DATA_BLOCK "S1.CABINET097.ALARM2"   // DB2589
// stored: AutoNumber true, DBAccessibleFromOPCUA true, DBAccessibleFromWebserver true, InstanceOfName BoolToUDInt_Inverted_Filtered, InstanceOfType FB
"BoolToUDInt_Inverted_Filtered "
BEGIN
END_DATA_BLOCK

DATA_BLOCK "S1.CABINET097.WARNING1"   // DB2590
// stored: AutoNumber true, DBAccessibleFromOPCUA true, DBAccessibleFromWebserver true, InstanceOfName BoolToUDInt_Inverted_Filtered, InstanceOfType FB
"BoolToUDInt_Inverted_Filtered "
BEGIN
END_DATA_BLOCK

DATA_BLOCK "S1.CABINET097.WARNING2"   // DB2591
// stored: AutoNumber true, DBAccessibleFromOPCUA true, DBAccessibleFromWebserver true, InstanceOfName BoolToUDInt_Inverted_Filtered, InstanceOfType FB
"BoolToUDInt_Inverted_Filtered "
BEGIN
END_DATA_BLOCK

DATA_BLOCK "S1.CABINET098.ALARM1"   // DB2592
// stored: AutoNumber true, DBAccessibleFromOPCUA true, DBAccessibleFromWebserver true, InstanceOfName BoolToUDInt_Inverted_Filtered, InstanceOfType FB
"BoolToUDInt_Inverted_Filtered "
BEGIN
END_DATA_BLOCK

DATA_BLOCK "S1.CABINET098.ALARM2"   // DB2593
// stored: AutoNumber true, DBAccessibleFromOPCUA true, DBAccessibleFromWebserver true, InstanceOfName BoolToUDInt_Inverted_Filtered, InstanceOfType FB
"BoolToUDInt_Inverted_Filtered "
BEGIN
END_DATA_BLOCK

DATA_BLOCK "S1.CABINET098.WARNING1"   // DB2594
// stored: AutoNumber true, DBAccessibleFromOPCUA true, DBAccessibleFromWebserver true, InstanceOfName BoolToUDInt_Inverted_Filtered, InstanceOfType FB
"BoolToUDInt_Inverted_Filtered "
BEGIN
END_DATA_BLOCK

DATA_BLOCK "S1.CABINET098.WARNING2"   // DB2595
// stored: AutoNumber true, DBAccessibleFromOPCUA true, DBAccessibleFromWebserver true, InstanceOfName BoolToUDInt_Inverted_Filtered, InstanceOfType FB
"BoolToUDInt_Inverted_Filtered "
BEGIN
END_DATA_BLOCK

DATA_BLOCK "S1.CABINET099.ALARM1"   // DB2596
// stored: AutoNumber true, DBAccessibleFromOPCUA true, DBAccessibleFromWebserver true, InstanceOfName BoolToUDInt_Inverted_Filtered, InstanceOfType FB
"BoolToUDInt_Inverted_Filtered "
BEGIN
END_DATA_BLOCK

DATA_BLOCK "S1.CABINET099.ALARM2"   // DB2597
// stored: AutoNumber true, DBAccessibleFromOPCUA true, DBAccessibleFromWebserver true, InstanceOfName BoolToUDInt_Inverted_Filtered, InstanceOfType FB
"BoolToUDInt_Inverted_Filtered "
BEGIN
END_DATA_BLOCK

DATA_BLOCK "S1.CABINET099.WARNING1"   // DB2598
// stored: AutoNumber true, DBAccessibleFromOPCUA true, DBAccessibleFromWebserver true, InstanceOfName BoolToUDInt_Inverted_Filtered, InstanceOfType FB
"BoolToUDInt_Inverted_Filtered "
BEGIN
END_DATA_BLOCK

DATA_BLOCK "S1.CABINET099.WARNING2"   // DB2599
// stored: AutoNumber true, DBAccessibleFromOPCUA true, DBAccessibleFromWebserver true, InstanceOfName BoolToUDInt_Inverted_Filtered, InstanceOfType FB
"BoolToUDInt_Inverted_Filtered "
BEGIN
END_DATA_BLOCK

DATA_BLOCK "S1.CABINET100.ALARM1"   // DB2600
// stored: AutoNumber true, DBAccessibleFromOPCUA true, DBAccessibleFromWebserver true, InstanceOfName BoolToUDInt_Inverted_Filtered, InstanceOfType FB
"BoolToUDInt_Inverted_Filtered "
BEGIN
END_DATA_BLOCK

DATA_BLOCK "S1.CABINET100.ALARM2"   // DB2601
// stored: AutoNumber true, DBAccessibleFromOPCUA true, DBAccessibleFromWebserver true, InstanceOfName BoolToUDInt_Inverted_Filtered, InstanceOfType FB
"BoolToUDInt_Inverted_Filtered "
BEGIN
END_DATA_BLOCK

DATA_BLOCK "S1.CABINET100.WARNING1"   // DB2602
// stored: AutoNumber true, DBAccessibleFromOPCUA true, DBAccessibleFromWebserver true, InstanceOfName BoolToUDInt_Inverted_Filtered, InstanceOfType FB
"BoolToUDInt_Inverted_Filtered "
BEGIN
END_DATA_BLOCK

DATA_BLOCK "S1.CABINET100.WARNING2"   // DB2603
// stored: AutoNumber true, DBAccessibleFromOPCUA true, DBAccessibleFromWebserver true, InstanceOfName BoolToUDInt_Inverted_Filtered, InstanceOfType FB
"BoolToUDInt_Inverted_Filtered "
BEGIN
END_DATA_BLOCK

DATA_BLOCK "S1.CABINET101.ALARM1"   // DB2604
// stored: AutoNumber true, DBAccessibleFromOPCUA true, DBAccessibleFromWebserver true, InstanceOfName BoolToUDInt_Inverted_Filtered, InstanceOfType FB
"BoolToUDInt_Inverted_Filtered "
BEGIN
END_DATA_BLOCK

DATA_BLOCK "S1.CABINET101.ALARM2"   // DB2605
// stored: AutoNumber true, DBAccessibleFromOPCUA true, DBAccessibleFromWebserver true, InstanceOfName BoolToUDInt_Inverted_Filtered, InstanceOfType FB
"BoolToUDInt_Inverted_Filtered "
BEGIN
END_DATA_BLOCK

DATA_BLOCK "S1.CABINET101.WARNING1"   // DB2606
// stored: AutoNumber true, DBAccessibleFromOPCUA true, DBAccessibleFromWebserver true, InstanceOfName BoolToUDInt_Inverted_Filtered, InstanceOfType FB
"BoolToUDInt_Inverted_Filtered "
BEGIN
END_DATA_BLOCK

DATA_BLOCK "S1.CABINET101.WARNING2"   // DB2607
// stored: AutoNumber true, DBAccessibleFromOPCUA true, DBAccessibleFromWebserver true, InstanceOfName BoolToUDInt_Inverted_Filtered, InstanceOfType FB
"BoolToUDInt_Inverted_Filtered "
BEGIN
END_DATA_BLOCK

DATA_BLOCK "S1.CABINET102.ALARM1"   // DB2608
// stored: AutoNumber true, DBAccessibleFromOPCUA true, DBAccessibleFromWebserver true, InstanceOfName BoolToUDInt_Inverted_Filtered, InstanceOfType FB
"BoolToUDInt_Inverted_Filtered "
BEGIN
END_DATA_BLOCK

DATA_BLOCK "S1.CABINET102.ALARM2"   // DB2609
// stored: AutoNumber true, DBAccessibleFromOPCUA true, DBAccessibleFromWebserver true, InstanceOfName BoolToUDInt_Inverted_Filtered, InstanceOfType FB
"BoolToUDInt_Inverted_Filtered "
BEGIN
END_DATA_BLOCK

DATA_BLOCK "S1.CABINET102.WARNING1"   // DB2610
// stored: AutoNumber true, DBAccessibleFromOPCUA true, DBAccessibleFromWebserver true, InstanceOfName BoolToUDInt_Inverted_Filtered, InstanceOfType FB
"BoolToUDInt_Inverted_Filtered "
BEGIN
END_DATA_BLOCK

DATA_BLOCK "S1.CABINET102.WARNING2"   // DB2611
// stored: AutoNumber true, DBAccessibleFromOPCUA true, DBAccessibleFromWebserver true, InstanceOfName BoolToUDInt_Inverted_Filtered, InstanceOfType FB
"BoolToUDInt_Inverted_Filtered "
BEGIN
END_DATA_BLOCK

DATA_BLOCK "S1.CABINET103.ALARM1"   // DB2612
// stored: AutoNumber true, DBAccessibleFromOPCUA true, DBAccessibleFromWebserver true, InstanceOfName BoolToUDInt_Inverted_Filtered, InstanceOfType FB
"BoolToUDInt_Inverted_Filtered "
BEGIN
END_DATA_BLOCK

DATA_BLOCK "S1.CABINET103.ALARM2"   // DB2613
// stored: AutoNumber true, DBAccessibleFromOPCUA true, DBAccessibleFromWebserver true, InstanceOfName BoolToUDInt_Inverted_Filtered, InstanceOfType FB
"BoolToUDInt_Inverted_Filtered "
BEGIN
END_DATA_BLOCK

DATA_BLOCK "S1.CABINET103.WARNING1"   // DB2614
// stored: AutoNumber true, DBAccessibleFromOPCUA true, DBAccessibleFromWebserver true, InstanceOfName BoolToUDInt_Inverted_Filtered, InstanceOfType FB
"BoolToUDInt_Inverted_Filtered "
BEGIN
END_DATA_BLOCK

DATA_BLOCK "S1.CABINET103.WARNING2"   // DB2615
// stored: AutoNumber true, DBAccessibleFromOPCUA true, DBAccessibleFromWebserver true, InstanceOfName BoolToUDInt_Inverted_Filtered, InstanceOfType FB
"BoolToUDInt_Inverted_Filtered "
BEGIN
END_DATA_BLOCK

DATA_BLOCK "S1.CABINET104.ALARM1"   // DB2616
// stored: AutoNumber true, DBAccessibleFromOPCUA true, DBAccessibleFromWebserver true, InstanceOfName BoolToUDInt_Inverted_Filtered, InstanceOfType FB
"BoolToUDInt_Inverted_Filtered "
BEGIN
END_DATA_BLOCK

DATA_BLOCK "S1.CABINET104.ALARM2"   // DB2617
// stored: AutoNumber true, DBAccessibleFromOPCUA true, DBAccessibleFromWebserver true, InstanceOfName BoolToUDInt_Inverted_Filtered, InstanceOfType FB
"BoolToUDInt_Inverted_Filtered "
BEGIN
END_DATA_BLOCK

DATA_BLOCK "S1.CABINET104.WARNING1"   // DB2618
// stored: AutoNumber true, DBAccessibleFromOPCUA true, DBAccessibleFromWebserver true, InstanceOfName BoolToUDInt_Inverted_Filtered, InstanceOfType FB
"BoolToUDInt_Inverted_Filtered "
BEGIN
END_DATA_BLOCK

DATA_BLOCK "S1.CABINET104.WARNING2"   // DB2619
// stored: AutoNumber true, DBAccessibleFromOPCUA true, DBAccessibleFromWebserver true, InstanceOfName BoolToUDInt_Inverted_Filtered, InstanceOfType FB
"BoolToUDInt_Inverted_Filtered "
BEGIN
END_DATA_BLOCK

DATA_BLOCK "S1.CABINET105.ALARM1"   // DB2620
// stored: AutoNumber true, DBAccessibleFromOPCUA true, DBAccessibleFromWebserver true, InstanceOfName BoolToUDInt_Inverted_Filtered, InstanceOfType FB
"BoolToUDInt_Inverted_Filtered "
BEGIN
END_DATA_BLOCK

DATA_BLOCK "S1.CABINET105.ALARM2"   // DB2621
// stored: AutoNumber true, DBAccessibleFromOPCUA true, DBAccessibleFromWebserver true, InstanceOfName BoolToUDInt_Inverted_Filtered, InstanceOfType FB
"BoolToUDInt_Inverted_Filtered "
BEGIN
END_DATA_BLOCK

DATA_BLOCK "S1.CABINET105.WARNING1"   // DB2622
// stored: AutoNumber true, DBAccessibleFromOPCUA true, DBAccessibleFromWebserver true, InstanceOfName BoolToUDInt_Inverted_Filtered, InstanceOfType FB
"BoolToUDInt_Inverted_Filtered "
BEGIN
END_DATA_BLOCK

DATA_BLOCK "S1.CABINET105.WARNING2"   // DB2623
// stored: AutoNumber true, DBAccessibleFromOPCUA true, DBAccessibleFromWebserver true, InstanceOfName BoolToUDInt_Inverted_Filtered, InstanceOfType FB
"BoolToUDInt_Inverted_Filtered "
BEGIN
END_DATA_BLOCK

DATA_BLOCK "S1.CABINET106.ALARM1"   // DB2624
// stored: AutoNumber true, DBAccessibleFromOPCUA true, DBAccessibleFromWebserver true, InstanceOfName BoolToUDInt_Inverted_Filtered, InstanceOfType FB
"BoolToUDInt_Inverted_Filtered "
BEGIN
END_DATA_BLOCK

DATA_BLOCK "S1.CABINET106.ALARM2"   // DB2625
// stored: AutoNumber true, DBAccessibleFromOPCUA true, DBAccessibleFromWebserver true, InstanceOfName BoolToUDInt_Inverted_Filtered, InstanceOfType FB
"BoolToUDInt_Inverted_Filtered "
BEGIN
END_DATA_BLOCK

DATA_BLOCK "S1.CABINET106.WARNING1"   // DB2626
// stored: AutoNumber true, DBAccessibleFromOPCUA true, DBAccessibleFromWebserver true, InstanceOfName BoolToUDInt_Inverted_Filtered, InstanceOfType FB
"BoolToUDInt_Inverted_Filtered "
BEGIN
END_DATA_BLOCK

DATA_BLOCK "S1.CABINET106.WARNING2"   // DB2627
// stored: AutoNumber true, DBAccessibleFromOPCUA true, DBAccessibleFromWebserver true, InstanceOfName BoolToUDInt_Inverted_Filtered, InstanceOfType FB
"BoolToUDInt_Inverted_Filtered "
BEGIN
END_DATA_BLOCK

DATA_BLOCK "S1.CABINET107.ALARM1"   // DB2628
// stored: AutoNumber true, DBAccessibleFromOPCUA true, DBAccessibleFromWebserver true, InstanceOfName BoolToUDInt_Inverted_Filtered, InstanceOfType FB
"BoolToUDInt_Inverted_Filtered "
BEGIN
END_DATA_BLOCK

DATA_BLOCK "S1.CABINET107.ALARM2"   // DB2629
// stored: AutoNumber true, DBAccessibleFromOPCUA true, DBAccessibleFromWebserver true, InstanceOfName BoolToUDInt_Inverted_Filtered, InstanceOfType FB
"BoolToUDInt_Inverted_Filtered "
BEGIN
END_DATA_BLOCK

DATA_BLOCK "S1.CABINET107.WARNING1"   // DB2630
// stored: AutoNumber true, DBAccessibleFromOPCUA true, DBAccessibleFromWebserver true, InstanceOfName BoolToUDInt_Inverted_Filtered, InstanceOfType FB
"BoolToUDInt_Inverted_Filtered "
BEGIN
END_DATA_BLOCK

DATA_BLOCK "S1.CABINET107.WARNING2"   // DB2631
// stored: AutoNumber true, DBAccessibleFromOPCUA true, DBAccessibleFromWebserver true, InstanceOfName BoolToUDInt_Inverted_Filtered, InstanceOfType FB
"BoolToUDInt_Inverted_Filtered "
BEGIN
END_DATA_BLOCK

DATA_BLOCK "S1.CABINET108.ALARM1"   // DB2632
// stored: AutoNumber true, DBAccessibleFromOPCUA true, DBAccessibleFromWebserver true, InstanceOfName BoolToUDInt_Inverted_Filtered, InstanceOfType FB
"BoolToUDInt_Inverted_Filtered "
BEGIN
END_DATA_BLOCK

DATA_BLOCK "S1.CABINET108.ALARM2"   // DB2633
// stored: AutoNumber true, DBAccessibleFromOPCUA true, DBAccessibleFromWebserver true, InstanceOfName BoolToUDInt_Inverted_Filtered, InstanceOfType FB
"BoolToUDInt_Inverted_Filtered "
BEGIN
END_DATA_BLOCK

DATA_BLOCK "S1.CABINET108.WARNING1"   // DB2634
// stored: AutoNumber true, DBAccessibleFromOPCUA true, DBAccessibleFromWebserver true, InstanceOfName BoolToUDInt_Inverted_Filtered, InstanceOfType FB
"BoolToUDInt_Inverted_Filtered "
BEGIN
END_DATA_BLOCK

DATA_BLOCK "S1.CABINET108.WARNING2"   // DB2635
// stored: AutoNumber true, DBAccessibleFromOPCUA true, DBAccessibleFromWebserver true, InstanceOfName BoolToUDInt_Inverted_Filtered, InstanceOfType FB
"BoolToUDInt_Inverted_Filtered "
BEGIN
END_DATA_BLOCK

DATA_BLOCK "S1.CABINET109.ALARM1"   // DB2636
// stored: AutoNumber true, DBAccessibleFromOPCUA true, DBAccessibleFromWebserver true, InstanceOfName BoolToUDInt_Inverted_Filtered, InstanceOfType FB
"BoolToUDInt_Inverted_Filtered "
BEGIN
END_DATA_BLOCK

DATA_BLOCK "S1.CABINET109.ALARM2"   // DB2637
// stored: AutoNumber true, DBAccessibleFromOPCUA true, DBAccessibleFromWebserver true, InstanceOfName BoolToUDInt_Inverted_Filtered, InstanceOfType FB
"BoolToUDInt_Inverted_Filtered "
BEGIN
END_DATA_BLOCK

DATA_BLOCK "S1.CABINET109.WARNING1"   // DB2638
// stored: AutoNumber true, DBAccessibleFromOPCUA true, DBAccessibleFromWebserver true, InstanceOfName BoolToUDInt_Inverted_Filtered, InstanceOfType FB
"BoolToUDInt_Inverted_Filtered "
BEGIN
END_DATA_BLOCK

DATA_BLOCK "S1.CABINET109.WARNING2"   // DB2639
// stored: AutoNumber true, DBAccessibleFromOPCUA true, DBAccessibleFromWebserver true, InstanceOfName BoolToUDInt_Inverted_Filtered, InstanceOfType FB
"BoolToUDInt_Inverted_Filtered "
BEGIN
END_DATA_BLOCK

DATA_BLOCK "S1.CABINET110.ALARM1"   // DB2640
// stored: AutoNumber true, DBAccessibleFromOPCUA true, DBAccessibleFromWebserver true, InstanceOfName BoolToUDInt_Inverted_Filtered, InstanceOfType FB
"BoolToUDInt_Inverted_Filtered "
BEGIN
END_DATA_BLOCK

DATA_BLOCK "S1.CABINET110.ALARM2"   // DB2641
// stored: AutoNumber true, DBAccessibleFromOPCUA true, DBAccessibleFromWebserver true, InstanceOfName BoolToUDInt_Inverted_Filtered, InstanceOfType FB
"BoolToUDInt_Inverted_Filtered "
BEGIN
END_DATA_BLOCK

DATA_BLOCK "S1.CABINET110.WARNING1"   // DB2642
// stored: AutoNumber true, DBAccessibleFromOPCUA true, DBAccessibleFromWebserver true, InstanceOfName BoolToUDInt_Inverted_Filtered, InstanceOfType FB
"BoolToUDInt_Inverted_Filtered "
BEGIN
END_DATA_BLOCK

DATA_BLOCK "S1.CABINET110.WARNING2"   // DB2643
// stored: AutoNumber true, DBAccessibleFromOPCUA true, DBAccessibleFromWebserver true, InstanceOfName BoolToUDInt_Inverted_Filtered, InstanceOfType FB
"BoolToUDInt_Inverted_Filtered "
BEGIN
END_DATA_BLOCK

DATA_BLOCK "S1.CABINET111.ALARM1"   // DB2644
// stored: AutoNumber true, DBAccessibleFromOPCUA true, DBAccessibleFromWebserver true, InstanceOfName BoolToUDInt_Inverted_Filtered, InstanceOfType FB
"BoolToUDInt_Inverted_Filtered "
BEGIN
END_DATA_BLOCK

DATA_BLOCK "S1.CABINET111.ALARM2"   // DB2645
// stored: AutoNumber true, DBAccessibleFromOPCUA true, DBAccessibleFromWebserver true, InstanceOfName BoolToUDInt_Inverted_Filtered, InstanceOfType FB
"BoolToUDInt_Inverted_Filtered "
BEGIN
END_DATA_BLOCK

DATA_BLOCK "S1.CABINET111.WARNING1"   // DB2646
// stored: AutoNumber true, DBAccessibleFromOPCUA true, DBAccessibleFromWebserver true, InstanceOfName BoolToUDInt_Inverted_Filtered, InstanceOfType FB
"BoolToUDInt_Inverted_Filtered "
BEGIN
END_DATA_BLOCK

DATA_BLOCK "S1.CABINET111.WARNING2"   // DB2647
// stored: AutoNumber true, DBAccessibleFromOPCUA true, DBAccessibleFromWebserver true, InstanceOfName BoolToUDInt_Inverted_Filtered, InstanceOfType FB
"BoolToUDInt_Inverted_Filtered "
BEGIN
END_DATA_BLOCK
